(*********************************** G.D S.p.A. - Technical Department ***********************************
============= PROGRAM INFO ============
FOLDER:             TBD
MACHINES INVOLVED:  TBD 

============= DESCRIPTION =============
csp machine declaration

============= REVISIONS ===============
Date		Version	 	Author      	Description             
----------	-------		------------  	--------------------------------------------
2019/04/05 	0000.00	 	M.Grasso		Creation of the PRG

**********************************************************************************************************)
(*$R process_ref := prc; $*)
PROGRAM csp_transfer_accumulator_finger_os
VAR
	
	prc:											process;
	prc_path:										STRING;
	
	axis:											axis;	
	servo_on_condition:								BOOL;
	axis_actual_position:							LREAL;

	case_presence_phasing_begin_window:				LREAL; (*$P unit := °; desc := Case presence phasing begin window; $*)
	case_presence_phasing_end_window:				LREAL; (*$P unit := °; desc := Case presence phasing end window; $*)
	case_presence_phasing:							BOOL; 	
	
	master_offset:									LREAL := 0;
	
	torque_limit:									INT := 500; (*$P $*)
	torque_limit_old:								INT;
	
	MOTOR_PHASE_VELOCITY_DEGPS:						LREAL := 90; (*$P $*)
	
	enable_delay: TON;
	Torque_force_constant: 							LREAL := 0.47;
END_VAR

VAR CONSTANT
	(*Just in case you prefer having constants instead of numbers*)
	MOTOR_MAX_VELOCITY_DEGPS:						LREAL := 9600;
	MOTOR_MAX_ACCELLERATION_DEGPS2:					LREAL := 4800;
	MOTOR_MAX_DECELLERATION_DEGPS2:					LREAL := 4800;
	MOTOR_MAX_JERK_DEGPS3:							LREAL := 100000000; 
	MOTOR_MAX_FOLLOWING_ERROR_DEG:					LREAL := 15;	//10/22/2021 PRS - increased from 5	
END_VAR

_read_var_input();

_object_manager();

IF 	NOT objects_running()
THEN
	RETURN;	
END_IF

_read_process_image();

_mode_manager();

CASE process_get_mode(prc) OF
	MODE_ABSENT:
		IF axis_get_mode(axis) = MODE_TEST
		THEN
			safety_integrated_series_close(csp_transfer_main_safety_drives_SD41200.chA_smes_sis);
		END_IF
		RETURN;
	MODE_INACTIVE:
		RETURN;
	MODE_TEST:
		_handle_process_test();
END_CASE

_set_runtime_properties();

(********************************* BODY *********************************)
axis.actual_torque := (axis.actual_current * Torque_force_constant)/1000;

// Sets torque Limit
IF torque_limit <> torque_limit_old
THEN
	 IF soe_drive_channel_write_parameter(
		channel:=csp_transfer_accumulator_finger_os.axis.soe_drive_channel, 
		idn:= S_0_IDN + 92, 
		data_element:=soe_drive_element_value , 
		data_source:= ADR(torque_limit), 
		data_lenght:= SIZEOF(torque_limit), 
		CONVERSION_this:= csp_transfer_accumulator_finger_os.axis.soe_drive^)= SOE_DRIVE_RETURN_VALUE_DONE
	THEN 
		Torque_limit_old := torque_limit;
	END_IF
END_IF


(************************************************************************)

_handle_messages();

_write_output();

ACTION _handle_messages:
;
END_ACTION

ACTION _handle_process_test:
;
END_ACTION

ACTION _mode_manager:
IF process_mode_req_is_pending(prc)
THEN
    process_apply_mode_req_first_step(prc);
    CASE process_get_mode(prc) OF
        MODE_TO_ABSENT:
			;
        MODE_TO_INACTIVE:
			;
        MODE_TO_TEST:
			;
        MODE_TO_OPERATIONAL:
			;
    END_CASE
    process_apply_mode_req_second_step(prc);
END_IF
END_ACTION

ACTION _object_manager:
IF objects_initialization()
THEN
	sub_process_init(
		object_name					:= 'csp_transfer_accumulator_finger_os.prc', 
		process						:= csp_transfer_accumulator_finger.prc, 
		CONVERSION_this				:= prc);
		
	prc_path 						:= process_get_path(prc);
	
	axis_init(
		object_name					:= CONCAT(prc_path, '_axis'), 
		axis_type					:= AXIS_TYPE_SERVO, 
		encoder_scaling_factor		:= G_SERVO_ENCODER_SCALING_FACTOR_DEGPINC,
		modulo						:= G_MODULO_360_DEG, 
		process						:= prc, 
		CONVERSION_this				:= axis);
		
	axis_init_absolute_encoder_preset(	
		position					:=	0,
		CONVERSION_this				:=	axis);	
	
	axis_set_max_dynamic(
		reference_velocity			:=	MOTOR_MAX_VELOCITY_DEGPS,
		velocity					:=	MOTOR_MAX_VELOCITY_DEGPS,
		acceleration				:=	MOTOR_MAX_ACCELLERATION_DEGPS2,
		deceleration				:=	MOTOR_MAX_DECELLERATION_DEGPS2,
		jerk						:=	MOTOR_MAX_JERK_DEGPS3,
		following_error				:=	MOTOR_MAX_FOLLOWING_ERROR_DEG,
		CONVERSION_this				:=	axis);
	
	jog_manager_add_axis(
		list_index					:= SMTR41203_TRANSFER_ACCUMULATOR_FINGER_OS,
		axis						:= axis,
		master_axis					:= FALSE,
		jog_type					:= JOG_TYPE_ROTATIVE,
		sw_limit_positive			:= 0.0,
		sw_limit_negative			:= 0.0,
		CONVERSION_this				:= csp_main_jogManager.jog_manager_real);

	axis_add_soe_drive(
		channel						:=	SOE_DRIVE_CHANNEL_A,
		soe_drive					:=	csp_transfer_main_drives.SD41200_drv,
		CONVERSION_this				:=	axis);

	IF 	csp_main_configurator.Physical_hw
	THEN
		axis_add_safety_integrated_series(
			safety_integrated_series := csp_transfer_main_safety_drives_SD41200.chA_smes_sis,
			CONVERSION_this			:= axis);
	END_IF
		
END_IF

IF objects_running()
THEN
	process_cycle(prc);
	axis_cycle(axis);
END_IF
END_ACTION

ACTION _read_process_image:
;
END_ACTION

ACTION _read_var_input:
;
END_ACTION

ACTION _set_runtime_properties:
axis_actual_position := axis_get_actual_modulo_position(axis);

enable_delay(IN:=axis_is_ready_to_enable(axis) , PT:=T#2S , Q=> servo_on_condition , ET=> );
	
IF 	(case_presence_phasing_begin_window <= case_presence_phasing_end_window)
THEN
	case_presence_phasing := 
		(axis_actual_position >= case_presence_phasing_begin_window) AND
		(axis_actual_position <= case_presence_phasing_end_window);
ELSE
	case_presence_phasing := 
		(axis_actual_position >= case_presence_phasing_begin_window) OR
		(axis_actual_position <= case_presence_phasing_end_window);
END_IF
END_ACTION

ACTION _write_output:
;
END_ACTION

END_PROGRAM

(* stored: Version 1.1.0.1, ProductVersion 3.1.4024.3
   POU csp_transfer_accumulator_finger_os: Id {409eee6f-3ea0-4940-acd1-c7922b4cbdd2}, SpecialFunc None
   Action _handle_messages: Id {318cb3c1-79f3-4bfc-8551-2056d31a543f}
   Action _handle_process_test: Id {2426949b-7b5e-44de-ae57-b4393dddfcc5}
   Action _mode_manager: Id {d5b640a5-269c-4cc8-a963-d4c03f43c3f2}
   Action _object_manager: Id {f75c72e2-3657-4056-b87c-de8add6b321f}
   Action _read_process_image: Id {6c59bae9-a77a-4a1d-a4ae-220f6aa32f5d}
   Action _read_var_input: Id {a5d7ac3c-26dc-45b9-b78d-fbe84d1e1799}
   Action _set_runtime_properties: Id {c93db77a-ee6c-44b0-8ff2-09a0b9ff85f8}
   Action _write_output: Id {b8c9b497-272b-403e-bfd5-2f111e596509} *)
